FUNCTION_BLOCK FB_Level3Handler IMPLEMENTS I_Handler
VAR_INPUT
END_VAR
VAR_OUTPUT
END_VAR
VAR
	_ipNextHandler		:I_Handler;
END_VAR

//FB_Init is always available implicitly and it is used primarily for initialization.
//The return value is not evaluated. For a specific influence, you can also declare the
//methods explicitly and provide additional code there with the standard initialization
//code. You can evaluate the return value.
METHOD FB_Init: BOOL
VAR_INPUT
    bInitRetains: BOOL; // TRUE: the retain variables are initialized (reset warm / reset cold)
    bInCopyCode: BOOL;  // TRUE: the instance will be copied to the copy code afterward (online change)   
	ipNextHandler	:I_Handler;
END_VAR
_ipNextHandler := ipNextHandler;
END_METHOD

METHOD handleRequest : BOOL
VAR_INPUT
	in_sRequest		: STRING;
END_VAR
IF FIND(in_sRequest, 'Level 3') <> 0 THEN
	ADSLOGSTR(msgCtrlMask:= ADSLOG_MSGTYPE_ERROR, msgFmtStr:= 'Request solved by Level 3. Request: %s', strArg:= in_sRequest);
ELSIF _ipNextHandler <> 0 THEN
	ADSLOGSTR(msgCtrlMask:= ADSLOG_MSGTYPE_ERROR, msgFmtStr:= 'Request cannot solved by Level 3.', strArg:= '');
	_ipNextHandler.handleRequest(in_sRequest);
ELSE
	ADSLOGSTR(msgCtrlMask:= ADSLOG_MSGTYPE_ERROR, msgFmtStr:= 'Request cannot solved by Level 3 and there is nobody else to pass it.', strArg:= '');	
END_IF
END_METHOD

END_FUNCTION_BLOCK

(* stored: Version 1.1.0.1
   POU FB_Level3Handler: Id {790ade86-5a34-4db8-b71c-c095ca8d7b26}, SpecialFunc None
   Method FB_Init: Id {a0e0ad6d-27f7-4b41-b43d-2cfe4b26a0f6}
   Method handleRequest: Id {92bd16dc-c683-460c-9c54-c46890ba9031} *)
